{attribute 'TcGenerated'}
{attribute 'no-analysis'}
{attribute 'linkalways'}
// This function has been automatically generated from the project information.
VAR_GLOBAL CONSTANT
    {attribute 'const_non_replaced'}
    stLibVersion_LCLS_Vacuum : ST_LibVersion := (iMajor := 2, iMinor := 6, iBuild := 6, iRevision := 0, nFlags := 1, sVersion := '2.6.6');
END_VAR

(* stored: Version 1.1.0.1
   GVL Global_Version: Id {cbc2521c-3dec-4c0c-84bb-251a510b24ad} *)
